(* PLC project v0.6.04_CycleSemiAuto.project, CODESYS CODESYS V3.5 SP19 Patch 1 *)
(* stored: creationDateTime 2026-08-17T05:53:47.247496, modificationDateTime 2026-08-17T05:53:47.247496 *)

TYPE ST_Chain_Winch_Safety : STRUCT
  Idx301_EmergencyChainClosed : BOOL;  (* 1 = Boucle Urgence OK (Armé) | 0 = Arrêt d'Urgence Appuyé 🔴 *)
  Idx302_SafeStopActive : BOOL;  (* 0 = Sain (Autorisé) | 1 = Arrêt Rapide Métier Actif 🔴 *)
  Idx303_PowerCutOffActive : BOOL;  (* 0 = Puissance OK | 1 = Coupure Puissance Sécurité 🔴 *)
  Idx304_TopSensorPhysical_DI : BOOL;  (* 1 = Capteur Haut Libre (Sain) | 0 = Butée Haute Atteinte 🔴 *)
  Idx305_TopSensorBypassActive : BOOL;  (* 0 = Capteur Actif | 1 = Capteur Haut Shunté IHM ⚠️ *)
  Idx306_AscentPermitEffective : BOOL;  (* 1 = Montée Autorisée | 0 = MONTÉE BLOQUÉE 🔴 *)
  Idx307_SlackCablePhysical_DI : BOOL;  (* 1 = Câble Tendu (Sain) | 0 = Mou de Câble Détecté 🔴 *)
  Idx308_SlackCableBypassActive : BOOL;  (* 0 = Capteur Actif | 1 = Mou de Câble Shunté IHM ⚠️ *)
  Idx309_DescendPermitEffective : BOOL;  (* 1 = Descente Autorisée | 0 = DESCENTE BLOQUÉE 🔴 *)
  Idx310_MecaFaultMask : WORD;  (* 0 = Pas de Défaut | >0 = Bitfield Défauts Méca A-E 🔴 *)
END_STRUCT;
END_TYPE
